FUNCTION_BLOCK ODriveCanSimpleTransporter
VAR_INPUT
END_VAR
VAR_OUTPUT
END_VAR
VAR
	_TxData AT%Q* : ST_CanQueue;
	_RxData AT%I* : ST_CanQueue;
	_bTxQueueNotEmpty : BOOL;
END_VAR

VAR_STAT CONSTANT
	_nMaxMsgCount : UINT := 10;
END_VAR

// Receive data cyclically
IF _TxData.RxCounter <> _RxData.RxCounter THEN
	_TxData.RxCounter := _RxData.RxCounter;
END_IF

// Send data if queue is not empty
_bTxQueueNotEmpty := _TxData.NoOfMessages <> 0;
SendCmd(bExecute:= _bTxQueueNotEmpty );

METHOD AddCmd
VAR_INPUT
	stCanMsg : ST_CanMessage;
END_VAR

VAR_OUTPUT
	//bBusy : BOOL;
	bError : BOOL;
	sErrorMsg : STRING;
	bDone : BOOL;
END_VAR
// Check if queue is fulled
IF _TxData.NoOfMessages >= _nMaxMsgCount THEN
	bError := TRUE;
	sErrorMsg := 'Tx message queue is fulled !';
	RETURN;
END_IF

// Count number of sent message
_TxData.NoOfMessages := _TxData.NoOfMessages + 1;

// Add message to queue (0-based)
_TxData.Messages[_TxData.NoOfMessages - 1] := stCanMsg;

bDone := TRUE;
END_METHOD

METHOD ReceiveData
VAR_INPUT
	nNodeId : UINT;
	eODriveCmd : E_ODriveCmd;
END_VAR

VAR_OUTPUT
	bExist : BOOL;
	stResultCanMsg : ST_CanMessage;
END_VAR

VAR
	nIdx : UINT;
	stCurCanMsg : ST_CanMessage;
	nCurNodeId : UINT;
	nCurCmd : UINT;
END_VAR
FOR nIdx := 0 TO (GVL_ODrive.nMaxMsgCount-1) DO
	
	// Parse data
	stCurCanMsg := _RxData.Messages[nIdx];
	nCurNodeId := SHR( (stCurCanMsg.CobId AND GVL_ODrive.nNodeId_Mask), GVL_ODrive.nNodeId_Shift );
	nCurCmd := SHR( (stCurCanMsg.CobId AND GVL_ODrive.nCmd_Mask), GVL_ODrive.nCmd_Shift );
	
	// Check if match input
	IF nNodeId <> nCurNodeId OR TO_UINT(eODriveCmd) <> nCurCmd THEN
		CONTINUE;
	END_IF
	
	bExist := TRUE;
	stResultCanMsg := stCurCanMsg;
	RETURN;
	
END_FOR
END_METHOD

METHOD PRIVATE SendCmd
VAR_INPUT
	bExecute : BOOL;
END_VAR
VAR_OUTPUT
	bBusy : BOOL;
	//bError : BOOL;
	bDone : BOOL;
END_VAR

VAR_INST
    nStep : UINT := 0;
END_VAR
CASE nStep OF
	0: // Idle
		IF bExecute THEN
			bBusy := TRUE;
			nStep := 1;
		END_IF
		
	1: // Send command
		_TxData.TxCounter := _TxData.TxCounter + 1;
		bBusy := TRUE;
		nStep := 2;
	
	2: // Check command sent
		IF _TxData.TxCounter = _RxData.TxCounter THEN
			_TxData.NoOfMessages := 0;	// Clear buffer count
			bDone := TRUE;
			nStep := 0;
		ELSE
			bBusy := TRUE;
		END_IF
		
END_CASE
END_METHOD

END_FUNCTION_BLOCK

(* stored: Version 1.1.0.1
   POU ODriveCanSimpleTransporter: Id {c60a47cd-3a50-4e37-b37f-89c661c67906}, SpecialFunc None
   Method AddCmd: Id {f539eac5-9aa6-44dc-ac60-e1b1afb830bb}
   Method ReceiveData: Id {f35617c3-1c7f-48a8-974c-4567958d847e}
   Method SendCmd: Id {114bb877-3e08-4fb7-a3e9-5688e34c6d83} *)
